// TwinCAT 3 PLC project MONETcommonTests
// Title: MONETcommonTests
// Company: IAG
// ProjectVersion: 0.1.0
// ProgramVersion: 3.1.4024.66
// libraries:
//   MONETcommon, * (IAG)
//   BROTLib, * (BROT)
//   HalfBROT, * (BROT)
//   AstroBROT, * (BROT)
//   Tc2_MC2, * (Beckhoff Automation GmbH)
//   Tc2_Standard, * (Beckhoff Automation GmbH)
//   Tc2_System, * (Beckhoff Automation GmbH)
//   Tc2_Utilities, * (Beckhoff Automation GmbH)
//   Tc3_Module, * (Beckhoff Automation GmbH)
//   VisuElemEventTable, 1.0.3.0 (System)
//   TcUnit, * (www.tcunit.org)
// project tree:
//   / PlcTask.TcTTO
//   POUs/ FB_NullComm.TcPOU, FB_MonetCoverControl_Tests.TcPOU, F_AzimuthOffsetOnAxis_Tests.TcPOU, MAIN.TcPOU
// real-time tasks:
//   TASK PlcTask: cycle T#10ms, priority 20, ADS port 350

CONFIGURATION MONETcommonTests
    RESOURCE PLC ON TwinCAT3
        TASK PlcTask(INTERVAL := T#10ms, PRIORITY := 20);
        PROGRAM MAIN WITH PlcTask : MAIN;
    END_RESOURCE
END_CONFIGURATION

// ---- POUs/MAIN.TcPOU
PROGRAM MAIN
VAR
	// TcUnit finds every FB_TestSuite instance by itself; it is enough to declare them here.
	fbCoverControlTests	: FB_MonetCoverControl_Tests;
	fbAzimuthOffsetTests	: F_AzimuthOffsetOnAxis_Tests;
END_VAR

TcUnit.RUN();

END_PROGRAM

// ---- POUs/FB_MonetCoverControl_Tests.TcPOU
// Tests for MONETcommon.FB_MonetCoverControl.
//
// IabCoverOpen/IabCoverClosed are AT%I* (hardware-mapped inside the FB itself), so a test running
// on a target with no linked EtherCAT hardware sees them default to FALSE. Both limit switches are
// wired "inverted" (abCoverOpen[i] := NOT IabCoverOpen[i]), so an unlinked/default-FALSE input
// reads as TRUE on both "open" and "closed" simultaneously -- this is itself the scenario that
// should raise bError (both switches active is treated as a limit-switch fault), independent of
// any command ever being issued.
FUNCTION_BLOCK FB_MonetCoverControl_Tests EXTENDS TcUnit.FB_TestSuite
VAR
END_VAR

Unlinked_Hardware_Reports_Error();

// On a target with no linked limit-switch hardware, both IabCoverOpen and IabCoverClosed default to
// FALSE, and the inverted polarity turns that into "both open and closed simultaneously" for every
// cover -- a real limit-switch-fault condition, not a test artifact. This anchors that FB_MonetCoverControl
// actually runs (compiles, instantiates, calls its own internal FBs) without any hardware or other
// MONETcommon/BROTLib dependency beyond I_Comm -- the open question flagged in the 2026-09-22
// add-tcunit-tests.md plan.
METHOD PRIVATE Unlinked_Hardware_Reports_Error
VAR
	fbComm	: FB_NullComm;
	fbCover	: MONETcommon.FB_MonetCoverControl(comm := fbComm);
END_VAR
TEST('Unlinked_Hardware_Reports_Error');
fbCover();
AssertTrue(Condition := fbCover.bError, Message := 'bError is TRUE with no limit-switch hardware linked');
TEST_FINISHED();
END_METHOD

END_FUNCTION_BLOCK

// ---- POUs/FB_NullComm.TcPOU
// Minimal I_Comm stub for tests: every Publish/PublishLog call is a no-op that reports success,
// so FBs under test can call fbComm.Publish(...) freely without a real MQTT connection.
FUNCTION_BLOCK FB_NullComm IMPLEMENTS BROTLib.I_Comm
VAR
END_VAR

METHOD Publish : BOOL
VAR_INPUT
	domain			: STRING(255) := 'environment';
	location		: STRING(255) := 'roof';
	parameter		: STRING(255);
	value			: STRING(255);
END_VAR
VAR_OUTPUT
	published	: BOOL;
END_VAR
Publish := TRUE;
published := TRUE;
END_METHOD

METHOD PublishLog : BOOL
VAR_INPUT
	level		: STRING(255) := 'INFO';
	message		: STRING(255);
END_VAR
VAR_OUTPUT
	published	: BOOL;
END_VAR
PublishLog := TRUE;
published := TRUE;
END_METHOD

END_FUNCTION_BLOCK

// ---- POUs/F_AzimuthOffsetOnAxis_Tests.TcPOU
// Tests for MONETcommon.F_AzimuthOffsetOnAxis, the azimuth offset bounded near the zenith (BROTLib#27).
FUNCTION_BLOCK F_AzimuthOffsetOnAxis_Tests EXTENDS TcUnit.FB_TestSuite
VAR
END_VAR

Horizon_Is_The_Offset_Itself();
Sixty_Degrees_Doubles();
Zenith_Is_Finite();
Result_Is_Limited_To_Ten_Degrees();

METHOD PRIVATE Horizon_Is_The_Offset_Itself
VAR
END_VAR
TEST('Horizon_Is_The_Offset_Itself');
AssertEquals_LREAL(Expected := 0.01, Actual := MONETcommon.F_AzimuthOffsetOnAxis(0.01, 0.0), Delta := 1.0E-12, Message := 'elevation 0');
TEST_FINISHED();
END_METHOD

// Below 89.5 deg the result is the plain offset / COS(elevation).
METHOD PRIVATE Sixty_Degrees_Doubles
VAR
END_VAR
TEST('Sixty_Degrees_Doubles');
AssertEquals_LREAL(Expected := 0.02, Actual := MONETcommon.F_AzimuthOffsetOnAxis(0.01, 60.0), Delta := 1.0E-12, Message := 'elevation 60');
AssertEquals_LREAL(Expected := -0.02, Actual := MONETcommon.F_AzimuthOffsetOnAxis(-0.01, 60.0), Delta := 1.0E-12, Message := 'elevation 60, negative offset');
AssertEquals_LREAL(Expected := 0.01 / COS(85.0 * 0.017453292519943295), Actual := MONETcommon.F_AzimuthOffsetOnAxis(0.01, 85.0), Delta := 1.0E-12, Message := 'elevation 85');
TEST_FINISHED();
END_METHOD

// At exactly 90 deg the old code divided by COS(90 deg) = 0 (up to rounding).
METHOD PRIVATE Zenith_Is_Finite
VAR
END_VAR
TEST('Zenith_Is_Finite');
AssertEquals_LREAL(Expected := 0.01 / 0.008726535498373935, Actual := MONETcommon.F_AzimuthOffsetOnAxis(0.01, 90.0), Delta := 1.0E-9, Message := 'elevation 90');
AssertEquals_LREAL(Expected := 0.01 / 0.008726535498373935, Actual := MONETcommon.F_AzimuthOffsetOnAxis(0.01, 89.9), Delta := 1.0E-9, Message := 'elevation 89.9');
TEST_FINISHED();
END_METHOD

METHOD PRIVATE Result_Is_Limited_To_Ten_Degrees
VAR
END_VAR
TEST('Result_Is_Limited_To_Ten_Degrees');
AssertEquals_LREAL(Expected := 10.0, Actual := MONETcommon.F_AzimuthOffsetOnAxis(1.0, 89.9), Delta := 1.0E-12, Message := 'positive');
AssertEquals_LREAL(Expected := -10.0, Actual := MONETcommon.F_AzimuthOffsetOnAxis(-1.0, 89.9), Delta := 1.0E-12, Message := 'negative');
AssertEquals_LREAL(Expected := 0.0, Actual := MONETcommon.F_AzimuthOffsetOnAxis(0.0, 90.0), Delta := 1.0E-12, Message := 'no offset at the zenith');
TEST_FINISHED();
END_METHOD

END_FUNCTION_BLOCK
